(* IEC 61131-3 sources: 1326_JeddahAppartment/1326 - Jeddah Appartment - Last/PLC2, 9 files *)

(* ---- PrgConnectHMIs.ST ---- *)
Type
  T_HMI_Info : struct
     SNo          : USINT;
     readStAdd    : UINT;
     writeStAdd   : UINT;
     readNoPoint  : UINT;
     writeNoPoint : UINT;
  End_Struct;

  //================= Read from HMI =================

  TShutterControl : struct
     Dw : WORD;
     UP : WORD;
  End_Struct;

  TFCU_Control : struct
     onOff       : WORD;
     SetTempCtrl : WORD; //  bit 0 for increment, bit 1 for decrement
     setTemp     : INT;
     fanSpeed    : WORD;
     mode        : WORD;
  End_Struct;

  T_HMI_DataRead : struct
     enLights   : Array[1..17] of WORD;
     enOutlets  : Array[1..8] of WORD;
     enShutters : Array[1..6] of TShutterControl;
     enFCUs     : Array[1..3] of TFCU_Control;
  End_Struct;

  //================= Write To HMI ==================

  TShutterStatus : struct
     Dw  : WORD;
     UP  : WORD;
     pos : WORD;
  End_Struct;

  TFCU_Status  : Struct
     onOffStatus    : WORD;
     setTemp        : INT;
     roomTemp       : INT;
     fanSpeed       : WORD;
     mode           : WORD;
     valve          : WORD;
     fanSpeedCtrl   : WORD;
     fanRotationVar : WORD;   // var for rotating the fan GIF in the HMI according to the current fan speed
  End_Struct;

  T_HMI_DataWrite : struct
     lightsStatus     : Array[1..17] of WORD;
     outletsStatus    : Array[1..8]  of WORD;
     motionSensStatus : Array[1..4]  of WORD;
     shuttersStatus   : Array[1..6]  of TShutterStatus;
     FCUs_Status      : Array[1..3]  of TFCU_Status;
  End_Struct;

End_Type

Var_Global Constant
   numOfHMIs : INT := 11;
End_Var

Var_Global Retain
   HMIs_DataRead  : Array[1..numOfHMIs] of T_HMI_DataRead;     // Data is read from HMI
   HMIs_DataWrite : Array[1..numOfHMIs] of T_HMI_DataWrite;    // Data is written to HMI

   HMIs_Info : Array[1..numOfHMIs] of T_HMI_Info := [()];
End_Var

Var_Global
  cmdArr : Array[1..numOfHMIs * 2] of TCmdStruct;
  GrSel  : USINT ;
End_Var

PROGRAM PrgConnectHMIs
  VAR_INPUT
  END_VAR
  VAR_OUTPUT
  END_VAR
  VAR
  master : fbModbusRTUmas2;
  //cmdArr : Array[1..numOfHMIs * 2] of TCmdStruct;

  i      : INT ;
  maxCmd : USINT;

  END_VAR
  VAR_TEMP
  END_VAR

  if IS_COLD_RESTART_PLC or IS_HOT_RESTART_PLC then
     GrSel := 2;
  end_if;

  for i := 1 to numOfHMIs do
      ModbusCmd(Gr := 2, SNo := HMIs_Info[i].SNo, FNC := 3,  StAdr := HMIs_Info[i].readStAdd,   NoPoint := HMIs_Info[i].readNoPoint, PtrData := adr(HMIs_DataRead[i]), Cmd := cmdArr[i*2-1]) ;

      ModbusCmd(Gr := 2, SNo := HMIs_Info[i].SNo, FNC := 16, StAdr := HMIs_Info[i].writeStAdd , NoPoint := HMIs_Info[i].writeNoPoint, PtrData := adr(HMIs_DataWrite[i]), Cmd := cmdArr[i*2]) ;
  end_for;

  //maxCmd := INT_TO_USINT(numOfHMIs * 2);

  maxCmd := 2;
  master(EN := true, GrSel := GrSel,  MaxCmd := maxCmd , chanCode := CH2_uni , Delay := T#0.2s, Commands := cmdArr[1], MBtimeOut := T#0.5s);

END_PROGRAM

(* ---- PrgDiningRoom.ST ---- *)
VAR_GLOBAL CONSTANT
   NumOfLightDiningRoom      : USINT := 5;
   NumOfOutletDiningRoom     : USINT := 2;
   NumOfCurtainDiningRoom    : USINT := 0;
   NumOfMotionSensDiningRoom : USINT := 1;
   NumOfFCUsDiningRoom       : USINT := 1;
   NumOfHMIsDiningRoom       : USINT := 2;
END_VAR

VAR_GLOBAL RETAIN
   lightsStatusDiningRoom  {PUBLIC_API} : TLightsStatus;
   outletsStatusDiningRoom {PUBLIC_API} : TOutletsStatus;
   setTempFCU_DiningRoom  : Array[1..NumOfFCUsDiningRoom] of REAL := [20];

END_VAR

PROGRAM PrgDiningRoom

  VAR
  //WebMaker
  lightsSelect   : BOOL;
  socketsSelect  : BOOL;
  shuttersSelect : BOOL;
  AC_Select      : BOOL;
  navSelect      : usint;

  //RCU
  RCU_ethAdr   : TRemoteEthAdr;
  RCU_IP : TIPadr := [192, 168, 0, 23];
  RCU_Ch_localPort : UINT;
  Set_IP           : BOOL;
  GetAllStatus  : BOOL;
  SendIamServer : BOOL;

  //controlRoom
  controlRoom   : fbControlRoom ;
  lightsOutputDevs     : TlightsOutputDevs     := [(DevAddress := 1 , loopAddress := 1),(DevAddress := 1 , loopAddress := 2),
                                                   (DevAddress := 1 , loopAddress := 3),(DevAddress := 1 , loopAddress := 4),
                                                   (DevAddress := 1 , loopAddress := 5)];

  outletOutputDevs     : ToutletOutputDevs     := [(DevAddress := 1 , loopAddress := 6),(DevAddress := 1 , loopAddress := 7)];

  (*curtainsUpOutputDevs : TcurtainsUpOutputDevs := [(DevAddress := 1 , loopAddress := 8)];
  curtainsDwOutputDevs : TcurtainsDwOutputDevs := [(DevAddress := 1 , loopAddress := 9)]; *)

  motionSensOutputDevs : TMotionSensOutputDevs := [(DevAddress := 1 , loopAddress := 1)];

  EnLights                            : TEnLights     ;
  EnLightsAN       {PUBLIC_API}       : TEnLightsAN   ;
  EnOutlets                           : TEnOutlets    ;
  EnOutletsAN      {PUBLIC_API}       : TEnOutletsAN  ;
  EnCurtainsUp     {PUBLIC_API}       : TEnCurtainsUp ;
  EnCurtainsDw     {PUBLIC_API}       : TEnCurtainsDW ;
   //EnLightsDiningRoomAN1  {PUBLIC_API}      : TEnLightsAN1    ;
   //stLightsDiningRoomAN  {PUBLIC_API}       : BOOL     ;
  //curtainsFB       : TCurtainsFB;
  //CurtainPositWm   : TCurtainPositWm;

  //
  enLights_RT  : Array[1..NumOfHMIsDiningRoom,1..NumOfLightDiningRoom] of R_TRIG;
  enLights_FT  : Array[1..NumOfHMIsDiningRoom,1..NumOfLightDiningRoom] of F_TRIG;

  enOutlets_RT : Array[1..NumOfHMIsDiningRoom,1..NumOfOutletDiningRoom] of R_TRIG;
  enOutlets_FT : Array[1..NumOfHMIsDiningRoom,1..NumOfOutletDiningRoom] of F_TRIG;

  (*
  enCurtainsUP_RT : Array[1..NumOfHMIsDiningRoom,1..NumOfCurtainDiningRoom] of R_TRIG;
  enCurtainsUP_FT : Array[1..NumOfHMIsDiningRoom,1..NumOfCurtainDiningRoom] of F_TRIG;

  enCurtainsDW_RT : Array[1..NumOfHMIsDiningRoom,1..NumOfCurtainDiningRoom] of R_TRIG;
  enCurtainsDW_FT : Array[1..NumOfHMIsDiningRoom,1..NumOfCurtainDiningRoom] of F_TRIG;
  *)

  //
  i , j : USINT;
  afterRestart_TP : TP;
  afterRestart_TP_FT : F_TRIG;

  //
  motionSensStatus                : TMotionSensStatus;
  CurtainsUpStatus   {PUBLIC_API} : TCurtainsUpStatus;
  CurtainsDwStatus   {PUBLIC_API} : TCurtainsDwStatus;

  // FCU VARS
  FCU          : Array[1..NumOfFCUsDiningRoom] of fbControlFCU;
  enableFCU    : Array[1..NumOfFCUsDiningRoom] of BOOL;
  settingsFCU  : Array[1..NumOfFCUsDiningRoom] of TFCU_Settings;

  //modeFCU      : Array[1..NumOfFCUsDiningRoom] of TFCU_Mode;
  //fanSpeedFCU  : Array[1..NumOfFCUsDiningRoom] of TFCU_FanSpeed;

  enFCUs_FT    : Array[1..NumOfHMIsDiningRoom,1..NumOfFCUsDiningRoom] of F_TRIG;
  enFCUs_RT    : Array[1..NumOfHMIsDiningRoom,1..NumOfFCUsDiningRoom] of R_TRIG;

  enFanHigh_RT : Array[1..NumOfHMIsDiningRoom,1..NumOfFCUsDiningRoom] of R_TRIG;
  enFanMed_RT  : Array[1..NumOfHMIsDiningRoom,1..NumOfFCUsDiningRoom] of R_TRIG;
  enFanLow_RT  : Array[1..NumOfHMIsDiningRoom,1..NumOfFCUsDiningRoom] of R_TRIG;
  enFanAuto_RT : Array[1..NumOfHMIsDiningRoom,1..NumOfFCUsDiningRoom] of R_TRIG;

  enFCUCool_RT    : Array[1..NumOfHMIsDiningRoom,1..NumOfFCUsDiningRoom] of R_TRIG;
  enFCUFanOnly_RT : Array[1..NumOfHMIsDiningRoom,1..NumOfFCUsDiningRoom] of R_TRIG;

  enSetTempIncr_RT : Array[1..NumOfHMIsDiningRoom,1..NumOfFCUsDiningRoom] of R_TRIG;
  enSetTempIncr_FT : Array[1..NumOfHMIsDiningRoom,1..NumOfFCUsDiningRoom] of F_TRIG;

  enSetTempDecr_RT : Array[1..NumOfHMIsDiningRoom,1..NumOfFCUsDiningRoom] of R_TRIG;
  enSetTempDecr_FT : Array[1..NumOfHMIsDiningRoom,1..NumOfFCUsDiningRoom] of F_TRIG;

  //HMIs[1..num
  HMI_Index : USINT;
  RCU_Index : USINT;
  HMI_Addresses : Array[1..NumOfHMIsDiningRoom] of USINT := [2, 10];

  END_VAR

   if navSelect = 0 then
     lightsSelect   := 1;
     socketsSelect  := 0;
     AC_Select      := 0;
  elsif navSelect = 1 then
     lightsSelect   := 0;
     socketsSelect  := 1;
     AC_Select      := 0;
  elsif navSelect = 2 then
     lightsSelect   := 0;
     socketsSelect  := 0;
     AC_Select      := 1;
  end_if;

  HMI_Index := 2;
  RCU_Index := 2;

  if GetRemoteIPaddress(chanCode := Eth1_uni1, ethAdr := RCU_ethAdr) then
     RCUs_IPs[RCU_Index] := RCU_ethAdr.remoteIP;
  end_if;

  HMIs_Info[HMI_Index].SNo := HMI_Addresses[1];
  HMIs_Info[HMI_Index].readStAdd  := 261;
  HMIs_Info[HMI_Index].writeStAdd := 321;
  HMIs_Info[HMI_Index].readNoPoint  := SIZEOF(HMIs_DataRead[HMI_Index]) / 2;
  HMIs_Info[HMI_Index].writeNoPoint := SIZEOF(HMIs_DataWrite[HMI_Index]) / 2;

  for i := 1 to NumOfHMIsDiningRoom-1 do
    HMIs_Info[HMI_Index+i] := HMIs_Info[HMI_Index];
    HMIs_Info[HMI_Index+i].SNo := HMI_Addresses[i+1];
  end_for;

  afterRestart_TP(IN := IS_COLD_RESTART_PLC or IS_HOT_RESTART_PLC, PT := T#2s );
  afterRestart_TP_FT(CLK := afterRestart_TP.Q);

  if afterRestart_TP_FT.Q then
     SendIamServer := 1;
  end_if;

  controlRoom(RCU_ChCode := ETH1_uni1 , RCU_PingDone := RCUs_PingDone[RCU_Index],
              numOfLights := NumOfLightDiningRoom , numOfOutlets := NumOfOutletDiningRoom , numOfCurtains := NumOfCurtainDiningRoom, numOfMotionSens := NumOfMotionSensDiningRoom,
              lightsOutputDevs := lightsOutputDevs , outletOutputDevs := outletOutputDevs ,
              RCU_CH_IN := void(ETH1_uni1_IN) , LightsStatus := lightsStatusDiningRoom ,OutletsStatus := outletsStatusDiningRoom, MotionSenStatus := motionSensStatus,
              EnLights := EnLights , EnLightsAN := EnLightsAN , EnOutlets := EnOutlets ,EnOutletsAN :=EnOutletsAN ,
              SendIamServer := SendIamServer , GetAllStatus := GetAllStatus);

              //stLightsDiningRoomAN := lightsStatusDiningRoom[1];

   FCU[1](enable := enableFCU[1], mode := settingsFCU[1].FCU_Mode, fanSpeed := settingsFCU[1].FCU_FanSpeed, setTemp := setTempFCU_DiningRoom[1], temp := FCU_Temp_DiningRoom, valve := FCU_valve_DiningRoom, fanLow := FCU_fanLow_DiningRoom,
                 fanMed := FCU_fanMed_DiningRoom, fanHigh := FCU_fanHigh_DiningRoom);

   for i := 1 to NumOfLightDiningRoom do
       HMIs_DataWrite[HMI_Index].lightsStatus[i] := BOOL_TO_WORD(lightsStatusDiningRoom[i]);
   end_for;

   for i := 1 to NumOfOutletDiningRoom do
       HMIs_DataWrite[HMI_Index].outletsStatus[i] := BOOL_TO_WORD(outletsStatusDiningRoom[i]);
   end_for;

   for i := 1 to NumOfMotionSensDiningRoom do
       HMIs_DataWrite[HMI_Index].motionSensStatus[i] := BOOL_TO_WORD(motionSensStatus[i]);
   end_for;

   for i := 1 to NumOfFCUsDiningRoom do
      HMIs_DataWrite[HMI_Index].FCUs_Status[i] := FCU[i].FCU_Status;
   end_for;

   for i := 1 to NumOfHMIsDiningRoom-1 do
     HMIs_DataWrite[HMI_Index+i] := HMIs_DataWrite[HMI_Index];
   end_for;

   for j := 1 to NumOfHMIsDiningRoom do
     for i := 1 to NumOfLightDiningRoom do

         enLights_RT[j,i](CLK := HMIs_DataRead[HMI_Index + j - 1].enLights[i]);

         enLights_FT[j,i](CLK := HMIs_DataRead[HMI_Index + j - 1].enLights[i]);

         if enLights_RT[j,i].Q or enLights_FT[j,i].Q then
            EnLights[i] := 1;
         end_if;
     end_for;
   end_for;

   for j := 1 to NumOfHMIsDiningRoom do
     for i := 1 to NumOfOutletDiningRoom do

         enOutlets_RT[j,i](CLK := HMIs_DataRead[HMI_Index + j - 1].enOutlets[i]);

         enOutlets_FT[j,i](CLK := HMIs_DataRead[HMI_Index + j - 1].enOutlets[i]);

         if enOutlets_RT[j,i].Q or enOutlets_FT[j,i].Q then
            EnOutlets[i] := 1;
         end_if;
     end_for;
   end_for;

  (*
   for j := 1 to NumOfHMIsDiningRoom do
     for i := 1 to NumOfCurtainDiningRoom do

         enCurtainsUP_RT[j,i](CLK := HMIs_DataRead[HMI_Index + j - 1].enShutters[i].UP.0);

         enCurtainsUP_FT[j,i](CLK := HMIs_DataRead[HMI_Index + j - 1].enShutters[i].UP.0);

         if enCurtainsUP_RT[j,i].Q or enCurtainsUP_FT[j,i].Q then
            EnCurtainsUp[i] := 1;
         end_if;

         enCurtainsDW_RT[j,i](CLK := HMIs_DataRead[HMI_Index + j - 1].enShutters[i].Dw.0);

         enCurtainsDW_FT[j,i](CLK := HMIs_DataRead[HMI_Index + j - 1].enShutters[i].Dw.0);

         if enCurtainsDW_RT[j,i].Q or enCurtainsDW_FT[j,i].Q then
            EnCurtainsDw[i] := 1;
         end_if;

     end_for;
   end_for;*)

   for j := 1 to NumOfHMIsDiningRoom do
      for i := 1 to NumOfFCUsDiningRoom do
          enFCUs_FT[j,i](CLK := HMIs_DataRead[HMI_Index + j - 1].enFCUs[i].onOff);
          enFCUs_RT[j,i](CLK := HMIs_DataRead[HMI_Index + j - 1].enFCUs[i].onOff);

          if enFCUs_FT[j,i].Q then
             enableFCU[i] := 0;
          end_if;
          if enFCUs_RT[j,i].Q then
             enableFCU[i] := 1;
          end_if;

          enFanAuto_RT[j,i](CLK := (HMIs_DataRead[HMI_Index + j - 1].enFCUs[i].fanSpeed = 8));
          enFanLow_RT[j,i](CLK := HMIs_DataRead[HMI_Index + j - 1].enFCUs[i].fanSpeed.0);
          enFanMed_RT[j,i](CLK := HMIs_DataRead[HMI_Index + j - 1].enFCUs[i].fanSpeed.1);
          enFanHigh_RT[j,i](CLK := HMIs_DataRead[HMI_Index + j - 1].enFCUs[i].fanSpeed.2);

          if enFanAuto_RT[j,i].Q then
             settingsFCU[i].FCU_FanSpeed := auto;
          end_if;
          if enFanLow_RT[j,i].Q then
             settingsFCU[i].FCU_FanSpeed := low;
          end_if;
          if enFanMed_RT[j,i].Q then
             settingsFCU[i].FCU_FanSpeed := med;
          end_if;
          if enFanHigh_RT[j,i].Q then
             settingsFCU[i].FCU_FanSpeed := high;
          end_if;

          enFCUCool_RT[j,i](CLK := (HMIs_DataRead[HMI_Index + j - 1].enFCUs[i].mode = 0));
          enFCUFanOnly_RT[j,i](CLK := HMIs_DataRead[HMI_Index + j - 1].enFCUs[i].mode.0);

          if enFCUCool_RT[j,i].Q then
             settingsFCU[i].FCU_Mode := cooling;
          end_if;
          if enFCUFanOnly_RT[j,i].Q then
             settingsFCU[i].FCU_Mode := fanOnly;
          end_if;

          enSetTempIncr_RT[j,i](CLK := HMIs_DataRead[HMI_Index + j - 1].enFCUs[i].SetTempCtrl.0);
          enSetTempIncr_FT[j,i](CLK := HMIs_DataRead[HMI_Index + j - 1].enFCUs[i].SetTempCtrl.0);

          if enSetTempIncr_RT[j,i].Q or enSetTempIncr_FT[j,i].Q then
             setTempFCU_DiningRoom[j] := setTempFCU_DiningRoom[j] + 0.5;
          end_if;

          enSetTempDecr_RT[j,i](CLK := HMIs_DataRead[HMI_Index + j - 1].enFCUs[i].SetTempCtrl.1);
          enSetTempDecr_FT[j,i](CLK := HMIs_DataRead[HMI_Index + j - 1].enFCUs[i].SetTempCtrl.1);

          if enSetTempDecr_RT[j,i].Q or enSetTempDecr_FT[j,i].Q then
             setTempFCU_DiningRoom[j] := setTempFCU_DiningRoom[j] - 0.5;
          end_if;

      end_for;
   end_for;

END_PROGRAM

(* ---- PrgInterance.ST ---- *)
VAR_GLOBAL CONSTANT
   NumOfLightInter    :USINT := 6;
   NumOfOutletInter   :USINT := 1;
   NumOfCurtainInter  :USINT := 0;
END_VAR

VAR_GLOBAL RETAIN
   lightsStatusInter  : TLightsStatus;
   outletsStatusInter : TOutletsStatus;
END_VAR

PROGRAM PrgInterance

  VAR
  //WebMaker
  lightsSelect   : BOOL;
  socketsSelect  : BOOL;
  navSelect      : usint;

  //RCU
  RCU_ethAdrToSet   : TRemoteEthAdr;
  RCU_IP : TIPadr := [192, 168, 0, 24];
  RCU_Ch_localPort : UINT;
  Set_IP           : BOOL;
  GetAllStatus  : BOOL;
  SendIamServer : BOOL;

  //controlRoom
 // controlRoom   : fbControlRoom ;
  lightsOutputDevs     : TlightsOutputDevs     := [(DevAddress := 1 , loopAddress := 1),(DevAddress := 1 , loopAddress := 2),
                                                   (DevAddress := 1 , loopAddress := 3),(DevAddress := 1 , loopAddress := 4),
                                                   (DevAddress := 1 , loopAddress := 5),(DevAddress := 1 , loopAddress := 6)];
  outletOutputDevs     : ToutletOutputDevs     := [(DevAddress := 1 , loopAddress := 7)];

  EnLights         : TEnLights     ;
  EnOutlets        : TEnOutlets    ;
  EnCurtainsUp     : TEnCurtainsUp ;
  EnCurtainsDw     : TEnCurtainsDW ;
  curtainsFB       : TCurtainsFB;
  CurtainsUpStatus : TCurtainsUpStatus;
  CurtainsDwStatus : TCurtainsDwStatus;
  END_VAR

  if navSelect = 0 then
     lightsSelect   := 1;
     socketsSelect  := 0;

  elsif navSelect = 1 then
     lightsSelect   := 0;
     socketsSelect  := 1;
  end_if;

  RCU_Ch_localPort := 61000;
  RCU_ethAdrToSet.remotePort := 3341;
  RCU_ethAdrToSet.localPort  := RCU_Ch_localPort;
  RCU_ethAdrToSet.remoteIP   := RCU_IP;

 (* controlRoom(RCU_ChCode := ETH1_uni0 , RCU_IP_toSet := RCU_IP, RCU_ethAdrToSet := RCU_ethAdrToSet ,
              numOfLights := NumOfLightInter , numOfOutlets := NumOfOutletInter , numOfCurtains := NumOfCurtainInter,
              lightsOutputDevs := lightsOutputDevs , outletOutputDevs := outletOutputDevs ,
              RCU_CH_IN := void(ETH1_uni0_IN) , LightsStatus := lightsStatusInter , OutletsStatus := outletsStatusInter,
              CurtainsUpStatus :=CurtainsUpStatus ,CurtainsDwStatus := CurtainsDwStatus ,CurtainsFB :=curtainsFB ,
              EnLights := EnLights , EnOutlets := EnOutlets ,EnCurtainsUp := EnCurtainsUp ,EnCurtainsDw :=EnCurtainsDw,
              SendIamServer := SendIamServer , GetAllStatus := GetAllStatus); *)
END_PROGRAM

(* ---- PrgKitchen.ST ---- *)
VAR_GLOBAL CONSTANT
   NumOfLightKitchen      : USINT := 4;
   NumOfOutletKitchen     : USINT := 5;
   NumOfCurtainKitchen    : USINT := 0;
   NumOfMotionSensKitchen : USINT := 1;
   NumOfFCUsKitchen       : USINT := 1;
   NumOfHMIsKitchen       : USINT := 1;
END_VAR

VAR_GLOBAL RETAIN
   lightsStatusKitchen  {PUBLIC_API} : TLightsStatus;
   outletsStatusKitchen {PUBLIC_API} : TOutletsStatus;
   setTempFCU_Kitchen  : Array[1..NumOfFCUsKitchen] of REAL := [20];

END_VAR

PROGRAM PrgKitchen

  VAR
  //WebMaker
  lightsSelect   : BOOL;
  socketsSelect  : BOOL;
  shuttersSelect : BOOL;
  AC_Select      : BOOL;
  navSelect      : usint;

  //RCU
  RCU_ethAdr   : TRemoteEthAdr;
  RCU_IP : TIPadr := [192, 168, 0, 23];
  RCU_Ch_localPort : UINT;
  Set_IP           : BOOL;
  GetAllStatus  : BOOL;
  SendIamServer : BOOL;

  //controlRoom
  controlRoom   : fbControlRoom ;
  lightsOutputDevs     : TlightsOutputDevs     := [(DevAddress := 1 , loopAddress := 1),(DevAddress := 1 , loopAddress := 2),
                                                   (DevAddress := 1 , loopAddress := 3),(DevAddress := 1 , loopAddress := 4)];

  outletOutputDevs     : ToutletOutputDevs     := [(DevAddress := 1 , loopAddress := 5),(DevAddress := 1 , loopAddress := 6),
                                                   (DevAddress := 1 , loopAddress := 7),(DevAddress := 1 , loopAddress := 8),(DevAddress := 1 , loopAddress := 9)];

  (*curtainsUpOutputDevs : TcurtainsUpOutputDevs := [(DevAddress := 1 , loopAddress := 8)];
  curtainsDwOutputDevs : TcurtainsDwOutputDevs := [(DevAddress := 1 , loopAddress := 9)]; *)

  motionSensOutputDevs : TMotionSensOutputDevs := [(DevAddress := 1 , loopAddress := 1)];

  EnLights                            : TEnLights     ;
  EnLightsAN       {PUBLIC_API}       : TEnLightsAN   ;
  EnOutlets                           : TEnOutlets    ;
  EnOutletsAN      {PUBLIC_API}       : TEnOutletsAN  ;
  EnCurtainsUp     {PUBLIC_API}       : TEnCurtainsUp ;
  EnCurtainsDw     {PUBLIC_API}       : TEnCurtainsDW ;
   //EnLightsKitchenAN1  {PUBLIC_API}      : TEnLightsAN1    ;
   //stLightsKitchenAN  {PUBLIC_API}       : BOOL     ;
  //curtainsFB       : TCurtainsFB;
  //CurtainPositWm   : TCurtainPositWm;

  //
  enLights_RT  : Array[1..NumOfHMIsKitchen,1..NumOfLightKitchen] of R_TRIG;
  enLights_FT  : Array[1..NumOfHMIsKitchen,1..NumOfLightKitchen] of F_TRIG;

  enOutlets_RT : Array[1..NumOfHMIsKitchen,1..NumOfOutletKitchen] of R_TRIG;
  enOutlets_FT : Array[1..NumOfHMIsKitchen,1..NumOfOutletKitchen] of F_TRIG;

  (*
  enCurtainsUP_RT : Array[1..NumOfHMIsKitchen,1..NumOfCurtainKitchen] of R_TRIG;
  enCurtainsUP_FT : Array[1..NumOfHMIsKitchen,1..NumOfCurtainKitchen] of F_TRIG;

  enCurtainsDW_RT : Array[1..NumOfHMIsKitchen,1..NumOfCurtainKitchen] of R_TRIG;
  enCurtainsDW_FT : Array[1..NumOfHMIsKitchen,1..NumOfCurtainKitchen] of F_TRIG;
  *)

  //
  i , j : USINT;
  afterRestart_TP : TP;
  afterRestart_TP_FT : F_TRIG;

  //
  motionSensStatus                : TMotionSensStatus;
  CurtainsUpStatus   {PUBLIC_API} : TCurtainsUpStatus;
  CurtainsDwStatus   {PUBLIC_API} : TCurtainsDwStatus;

  // FCU VARS
  FCU          : Array[1..NumOfFCUsKitchen] of fbControlFCU;
  enableFCU    : Array[1..NumOfFCUsKitchen] of BOOL;
  settingsFCU  : Array[1..NumOfFCUsKitchen] of TFCU_Settings;

  //modeFCU      : Array[1..NumOfFCUsKitchen] of TFCU_Mode;
  //fanSpeedFCU  : Array[1..NumOfFCUsKitchen] of TFCU_FanSpeed;

  enFCUs_FT    : Array[1..NumOfHMIsKitchen,1..NumOfFCUsKitchen] of F_TRIG;
  enFCUs_RT    : Array[1..NumOfHMIsKitchen,1..NumOfFCUsKitchen] of R_TRIG;

  enFanHigh_RT : Array[1..NumOfHMIsKitchen,1..NumOfFCUsKitchen] of R_TRIG;
  enFanMed_RT  : Array[1..NumOfHMIsKitchen,1..NumOfFCUsKitchen] of R_TRIG;
  enFanLow_RT  : Array[1..NumOfHMIsKitchen,1..NumOfFCUsKitchen] of R_TRIG;
  enFanAuto_RT : Array[1..NumOfHMIsKitchen,1..NumOfFCUsKitchen] of R_TRIG;

  enFCUCool_RT    : Array[1..NumOfHMIsKitchen,1..NumOfFCUsKitchen] of R_TRIG;
  enFCUFanOnly_RT : Array[1..NumOfHMIsKitchen,1..NumOfFCUsKitchen] of R_TRIG;

  enSetTempIncr_RT : Array[1..NumOfHMIsKitchen,1..NumOfFCUsKitchen] of R_TRIG;
  enSetTempIncr_FT : Array[1..NumOfHMIsKitchen,1..NumOfFCUsKitchen] of F_TRIG;

  enSetTempDecr_RT : Array[1..NumOfHMIsKitchen,1..NumOfFCUsKitchen] of R_TRIG;
  enSetTempDecr_FT : Array[1..NumOfHMIsKitchen,1..NumOfFCUsKitchen] of F_TRIG;

  //HMIs[1..num
  HMI_Index : USINT;
  RCU_Index : USINT;
  HMI_Addresses : Array[1..NumOfHMIsKitchen] of USINT := [7];

  END_VAR

     if navSelect = 0 then
     lightsSelect   := 1;
     socketsSelect  := 0;
     AC_Select      := 0;
  elsif navSelect = 1 then
     lightsSelect   := 0;
     socketsSelect  := 1;
     AC_Select      := 0;
  elsif navSelect = 2 then
     lightsSelect   := 0;
     socketsSelect  := 0;
     AC_Select      := 1;
  end_if;

  HMI_Index := 6;
  RCU_Index := 4;

  if GetRemoteIPaddress(chanCode := Eth1_uni3, ethAdr := RCU_ethAdr) then
     RCUs_IPs[RCU_Index] := RCU_ethAdr.remoteIP;
  end_if;

  HMIs_Info[HMI_Index].SNo := HMI_Addresses[1];
  HMIs_Info[HMI_Index].readStAdd  := 521;
  HMIs_Info[HMI_Index].writeStAdd := 581;
  HMIs_Info[HMI_Index].readNoPoint  := SIZEOF(HMIs_DataRead[HMI_Index]) / 2;
  HMIs_Info[HMI_Index].writeNoPoint := SIZEOF(HMIs_DataWrite[HMI_Index]) / 2;

  for i := 1 to NumOfHMIsKitchen-1 do
    HMIs_Info[HMI_Index+i] := HMIs_Info[HMI_Index];
    HMIs_Info[HMI_Index+i].SNo := HMI_Addresses[i+1];
  end_for;

  afterRestart_TP(IN := IS_COLD_RESTART_PLC or IS_HOT_RESTART_PLC, PT := T#2s );
  afterRestart_TP_FT(CLK := afterRestart_TP.Q);

  if afterRestart_TP_FT.Q then
     SendIamServer := 1;
  end_if;

  controlRoom(RCU_ChCode := ETH1_uni3 , RCU_PingDone := RCUs_PingDone[RCU_Index],
              numOfLights := NumOfLightKitchen , numOfOutlets := NumOfOutletKitchen , numOfCurtains := NumOfCurtainKitchen, numOfMotionSens := NumOfMotionSensKitchen,
              lightsOutputDevs := lightsOutputDevs , outletOutputDevs := outletOutputDevs ,
              RCU_CH_IN := void(ETH1_uni3_IN) , LightsStatus := lightsStatusKitchen ,OutletsStatus := outletsStatusKitchen, MotionSenStatus := motionSensStatus,
              EnLights := EnLights , EnLightsAN := EnLightsAN , EnOutlets := EnOutlets ,EnOutletsAN :=EnOutletsAN ,
              SendIamServer := SendIamServer , GetAllStatus := GetAllStatus);

              //stLightsKitchenAN := lightsStatusKitchen[1];

   FCU[1](enable := enableFCU[1], mode := settingsFCU[1].FCU_Mode, fanSpeed := settingsFCU[1].FCU_FanSpeed, setTemp := setTempFCU_Kitchen[1], temp := FCU_Temp_Kitchen, valve := FCU_valve_Kitchen, fanLow := FCU_fanLow_Kitchen,
                 fanMed := FCU_fanMed_Kitchen, fanHigh := FCU_fanHigh_Kitchen);

   for i := 1 to NumOfLightKitchen do
       HMIs_DataWrite[HMI_Index].lightsStatus[i] := BOOL_TO_WORD(lightsStatusKitchen[i]);
   end_for;

   for i := 1 to NumOfOutletKitchen do
       HMIs_DataWrite[HMI_Index].outletsStatus[i] := BOOL_TO_WORD(outletsStatusKitchen[i]);
   end_for;

   for i := 1 to NumOfMotionSensKitchen do
       HMIs_DataWrite[HMI_Index].motionSensStatus[i] := BOOL_TO_WORD(motionSensStatus[i]);
   end_for;

   for i := 1 to NumOfFCUsKitchen do
      HMIs_DataWrite[HMI_Index].FCUs_Status[i] := FCU[i].FCU_Status;
   end_for;

   for i := 1 to NumOfHMIsKitchen-1 do
     HMIs_DataWrite[HMI_Index+i] := HMIs_DataWrite[HMI_Index];
   end_for;

   for j := 1 to NumOfHMIsKitchen do
     for i := 1 to NumOfLightKitchen do

         enLights_RT[j,i](CLK := HMIs_DataRead[HMI_Index + j - 1].enLights[i]);

         enLights_FT[j,i](CLK := HMIs_DataRead[HMI_Index + j - 1].enLights[i]);

         if enLights_RT[j,i].Q or enLights_FT[j,i].Q then
            EnLights[i] := 1;
         end_if;
     end_for;
   end_for;

   for j := 1 to NumOfHMIsKitchen do
     for i := 1 to NumOfOutletKitchen do

         enOutlets_RT[j,i](CLK := HMIs_DataRead[HMI_Index + j - 1].enOutlets[i]);

         enOutlets_FT[j,i](CLK := HMIs_DataRead[HMI_Index + j - 1].enOutlets[i]);

         if enOutlets_RT[j,i].Q or enOutlets_FT[j,i].Q then
            EnOutlets[i] := 1;
         end_if;
     end_for;
   end_for;

  (*
   for j := 1 to NumOfHMIsKitchen do
     for i := 1 to NumOfCurtainKitchen do

         enCurtainsUP_RT[j,i](CLK := HMIs_DataRead[HMI_Index + j - 1].enShutters[i].UP.0);

         enCurtainsUP_FT[j,i](CLK := HMIs_DataRead[HMI_Index + j - 1].enShutters[i].UP.0);

         if enCurtainsUP_RT[j,i].Q or enCurtainsUP_FT[j,i].Q then
            EnCurtainsUp[i] := 1;
         end_if;

         enCurtainsDW_RT[j,i](CLK := HMIs_DataRead[HMI_Index + j - 1].enShutters[i].Dw.0);

         enCurtainsDW_FT[j,i](CLK := HMIs_DataRead[HMI_Index + j - 1].enShutters[i].Dw.0);

         if enCurtainsDW_RT[j,i].Q or enCurtainsDW_FT[j,i].Q then
            EnCurtainsDw[i] := 1;
         end_if;

     end_for;
   end_for;*)

   for j := 1 to NumOfHMIsKitchen do
      for i := 1 to NumOfFCUsKitchen do
          enFCUs_FT[j,i](CLK := HMIs_DataRead[HMI_Index + j - 1].enFCUs[i].onOff);
          enFCUs_RT[j,i](CLK := HMIs_DataRead[HMI_Index + j - 1].enFCUs[i].onOff);

          if enFCUs_FT[j,i].Q then
             enableFCU[i] := 0;
          end_if;
          if enFCUs_RT[j,i].Q then
             enableFCU[i] := 1;
          end_if;

          enFanAuto_RT[j,i](CLK := (HMIs_DataRead[HMI_Index + j - 1].enFCUs[i].fanSpeed = 8));
          enFanLow_RT[j,i](CLK := HMIs_DataRead[HMI_Index + j - 1].enFCUs[i].fanSpeed.0);
          enFanMed_RT[j,i](CLK := HMIs_DataRead[HMI_Index + j - 1].enFCUs[i].fanSpeed.1);
          enFanHigh_RT[j,i](CLK := HMIs_DataRead[HMI_Index + j - 1].enFCUs[i].fanSpeed.2);

          if enFanAuto_RT[j,i].Q then
             settingsFCU[i].FCU_FanSpeed := auto;
          end_if;
          if enFanLow_RT[j,i].Q then
             settingsFCU[i].FCU_FanSpeed := low;
          end_if;
          if enFanMed_RT[j,i].Q then
             settingsFCU[i].FCU_FanSpeed := med;
          end_if;
          if enFanHigh_RT[j,i].Q then
             settingsFCU[i].FCU_FanSpeed := high;
          end_if;

          enFCUCool_RT[j,i](CLK := (HMIs_DataRead[HMI_Index + j - 1].enFCUs[i].mode = 0));
          enFCUFanOnly_RT[j,i](CLK := HMIs_DataRead[HMI_Index + j - 1].enFCUs[i].mode.0);

          if enFCUCool_RT[j,i].Q then
             settingsFCU[i].FCU_Mode := cooling;
          end_if;
          if enFCUFanOnly_RT[j,i].Q then
             settingsFCU[i].FCU_Mode := fanOnly;
          end_if;

          enSetTempIncr_RT[j,i](CLK := HMIs_DataRead[HMI_Index + j - 1].enFCUs[i].SetTempCtrl.0);
          enSetTempIncr_FT[j,i](CLK := HMIs_DataRead[HMI_Index + j - 1].enFCUs[i].SetTempCtrl.0);

          if enSetTempIncr_RT[j,i].Q or enSetTempIncr_FT[j,i].Q then
             setTempFCU_Kitchen[j] := setTempFCU_Kitchen[j] + 0.5;
          end_if;

          enSetTempDecr_RT[j,i](CLK := HMIs_DataRead[HMI_Index + j - 1].enFCUs[i].SetTempCtrl.1);
          enSetTempDecr_FT[j,i](CLK := HMIs_DataRead[HMI_Index + j - 1].enFCUs[i].SetTempCtrl.1);

          if enSetTempDecr_RT[j,i].Q or enSetTempDecr_FT[j,i].Q then
             setTempFCU_Kitchen[j] := setTempFCU_Kitchen[j] - 0.5;
          end_if;

      end_for;
   end_for;

END_PROGRAM

(* ---- PrgLivingRoom.ST ---- *)
VAR_GLOBAL CONSTANT
   NumOfLightLivingRoom      : USINT := 5;
   NumOfOutletLivingRoom     : USINT := 2;
   NumOfCurtainLivingRoom    : USINT := 2;
   NumOfMotionSensLivingRoom : USINT := 1;
   NumOfFCUsLivingRoom       : USINT := 0;
   NumOfHMIsLivingRoom       : USINT := 2;
END_VAR

VAR_GLOBAL RETAIN
   lightsStatusLivingRoom  {PUBLIC_API} : TLightsStatus;
   outletsStatusLivingRoom {PUBLIC_API} : TOutletsStatus;
  // setTempFCU_LivingRoom  : Array[1..NumOfFCUsLivingRoom] of REAL := [20];

END_VAR

PROGRAM PrgLivingRoom

  VAR
  //WebMaker
  lightsSelect   : BOOL;
  socketsSelect  : BOOL;
  shuttersSelect : BOOL;
  AC_Select      : BOOL;
  navSelect      : usint;

  //RCU
  RCU_ethAdr   : TRemoteEthAdr;
  RCU_IP : TIPadr := [192, 168, 0, 23];
  RCU_Ch_localPort : UINT;
  Set_IP           : BOOL;
  GetAllStatus  : BOOL;
  SendIamServer : BOOL;

  //controlRoom
  controlRoom   : fbControlRoom ;
  lightsOutputDevs     : TlightsOutputDevs     := [(DevAddress := 1 , loopAddress := 1),(DevAddress := 1 , loopAddress := 2),
                                                   (DevAddress := 1 , loopAddress := 3),(DevAddress := 1 , loopAddress := 4),
                                                   (DevAddress := 1 , loopAddress := 5)];

  outletOutputDevs     : ToutletOutputDevs     := [(DevAddress := 1 , loopAddress := 6),(DevAddress := 1 , loopAddress := 7)];

  curtainsUpOutputDevs : TcurtainsUpOutputDevs := [(DevAddress := 2 , loopAddress := 1), (DevAddress := 2 , loopAddress := 3)];
  curtainsDwOutputDevs : TcurtainsDwOutputDevs := [(DevAddress := 2 , loopAddress := 2), (DevAddress := 2 , loopAddress := 4)];

  motionSensOutputDevs : TMotionSensOutputDevs := [(DevAddress := 1 , loopAddress := 1)];

  EnLights                            : TEnLights     ;
  EnLightsAN       {PUBLIC_API}       : TEnLightsAN   ;
  EnOutlets                           : TEnOutlets    ;
  EnOutletsAN      {PUBLIC_API}       : TEnOutletsAN  ;
  EnCurtainsUp     {PUBLIC_API}       : TEnCurtainsUp ;
  EnCurtainsDw     {PUBLIC_API}       : TEnCurtainsDW ;
   //EnLightsLivingRoomAN1  {PUBLIC_API}      : TEnLightsAN1    ;
   //stLightsLivingRoomAN  {PUBLIC_API}       : BOOL     ;
  //curtainsFB       : TCurtainsFB;
  //CurtainPositWm   : TCurtainPositWm;

  //
  enLights_RT  : Array[1..NumOfHMIsLivingRoom,1..NumOfLightLivingRoom] of R_TRIG;
  enLights_FT  : Array[1..NumOfHMIsLivingRoom,1..NumOfLightLivingRoom] of F_TRIG;

  enOutlets_RT : Array[1..NumOfHMIsLivingRoom,1..NumOfOutletLivingRoom] of R_TRIG;
  enOutlets_FT : Array[1..NumOfHMIsLivingRoom,1..NumOfOutletLivingRoom] of F_TRIG;

  enCurtainsUP_RT : Array[1..NumOfHMIsLivingRoom,1..NumOfCurtainLivingRoom] of R_TRIG;
  enCurtainsUP_FT : Array[1..NumOfHMIsLivingRoom,1..NumOfCurtainLivingRoom] of F_TRIG;

  enCurtainsDW_RT : Array[1..NumOfHMIsLivingRoom,1..NumOfCurtainLivingRoom] of R_TRIG;
  enCurtainsDW_FT : Array[1..NumOfHMIsLivingRoom,1..NumOfCurtainLivingRoom] of F_TRIG;

  //
  i , j : USINT;
  afterRestart_TP : TP;
  afterRestart_TP_FT : F_TRIG;

  //
  motionSensStatus                : TMotionSensStatus;
  CurtainsUpStatus   {PUBLIC_API} : TCurtainsUpStatus;
  CurtainsDwStatus   {PUBLIC_API} : TCurtainsDwStatus;

  // FCU VARS
 (* FCU          : Array[1..NumOfFCUsLivingRoom] of fbControlFCU;
  enableFCU    : Array[1..NumOfFCUsLivingRoom] of BOOL;
  settingsFCU  : Array[1..NumOfFCUsLivingRoom] of TFCU_Settings;

  //modeFCU      : Array[1..NumOfFCUsLivingRoom] of TFCU_Mode;
  //fanSpeedFCU  : Array[1..NumOfFCUsLivingRoom] of TFCU_FanSpeed;

  enFCUs_FT    : Array[1..NumOfHMIsLivingRoom,1..NumOfFCUsLivingRoom] of F_TRIG;
  enFCUs_RT    : Array[1..NumOfHMIsLivingRoom,1..NumOfFCUsLivingRoom] of R_TRIG;

  enFanHigh_RT : Array[1..NumOfHMIsLivingRoom,1..NumOfFCUsLivingRoom] of R_TRIG;
  enFanMed_RT  : Array[1..NumOfHMIsLivingRoom,1..NumOfFCUsLivingRoom] of R_TRIG;
  enFanLow_RT  : Array[1..NumOfHMIsLivingRoom,1..NumOfFCUsLivingRoom] of R_TRIG;
  enFanAuto_RT : Array[1..NumOfHMIsLivingRoom,1..NumOfFCUsLivingRoom] of R_TRIG;

  enFCUCool_RT    : Array[1..NumOfHMIsLivingRoom,1..NumOfFCUsLivingRoom] of R_TRIG;
  enFCUFanOnly_RT : Array[1..NumOfHMIsLivingRoom,1..NumOfFCUsLivingRoom] of R_TRIG;

  enSetTempIncr_RT : Array[1..NumOfHMIsLivingRoom,1..NumOfFCUsLivingRoom] of R_TRIG;
  enSetTempIncr_FT : Array[1..NumOfHMIsLivingRoom,1..NumOfFCUsLivingRoom] of F_TRIG;

  enSetTempDecr_RT : Array[1..NumOfHMIsLivingRoom,1..NumOfFCUsLivingRoom] of R_TRIG;
  enSetTempDecr_FT : Array[1..NumOfHMIsLivingRoom,1..NumOfFCUsLivingRoom] of F_TRIG;  *)

  //HMIs[1..num
  HMI_Index : USINT;
  RCU_Index : USINT;
  HMI_Addresses : Array[1..NumOfHMIsLivingRoom] of USINT := [3, 5];

  END_VAR

   if navSelect = 0 then
     lightsSelect   := 1;
     socketsSelect  := 0;
     shuttersSelect := 0;
  elsif navSelect = 1 then
     lightsSelect   := 0;
     socketsSelect  := 1;
     shuttersSelect := 0;
  elsif navSelect = 2 then
     lightsSelect   := 0;
     socketsSelect  := 0;
     shuttersSelect := 1;
  end_if;

  HMI_Index := 4;
  RCU_Index := 3;

  if GetRemoteIPaddress(chanCode := Eth1_uni2, ethAdr := RCU_ethAdr) then
     RCUs_IPs[RCU_Index] := RCU_ethAdr.remoteIP;
  end_if;

  HMIs_Info[HMI_Index].SNo := HMI_Addresses[1];
  HMIs_Info[HMI_Index].readStAdd  := 391;
  HMIs_Info[HMI_Index].writeStAdd := 451;
  HMIs_Info[HMI_Index].readNoPoint  := SIZEOF(HMIs_DataRead[HMI_Index]) / 2;
  HMIs_Info[HMI_Index].writeNoPoint := SIZEOF(HMIs_DataWrite[HMI_Index]) / 2;

  for i := 1 to NumOfHMIsLivingRoom-1 do
    HMIs_Info[HMI_Index+i] := HMIs_Info[HMI_Index];
    HMIs_Info[HMI_Index+i].SNo := HMI_Addresses[i+1];
  end_for;

  afterRestart_TP(IN := IS_COLD_RESTART_PLC or IS_HOT_RESTART_PLC, PT := T#2s );
  afterRestart_TP_FT(CLK := afterRestart_TP.Q);

  if afterRestart_TP_FT.Q then
     SendIamServer := 1;
  end_if;

  controlRoom(RCU_ChCode := ETH1_uni2 , RCU_PingDone := RCUs_PingDone[RCU_Index],
              numOfLights := NumOfLightLivingRoom , numOfOutlets := NumOfOutletLivingRoom , numOfCurtains := NumOfCurtainLivingRoom, numOfMotionSens := NumOfMotionSensLivingRoom,
              lightsOutputDevs := lightsOutputDevs , outletOutputDevs := outletOutputDevs ,
              curtainsUpOutputDevs := curtainsUpOutputDevs , curtainsDwOutputDevs := curtainsDwOutputDevs,
              RCU_CH_IN := void(ETH1_uni2_IN) , LightsStatus := lightsStatusLivingRoom ,OutletsStatus := outletsStatusLivingRoom, MotionSenStatus := motionSensStatus,
              EnLights := EnLights , EnLightsAN := EnLightsAN , EnOutlets := EnOutlets ,EnOutletsAN :=EnOutletsAN ,
              SendIamServer := SendIamServer , GetAllStatus := GetAllStatus);

              //stLightsLivingRoomAN := lightsStatusLivingRoom[1];

  (* FCU[1](enable := enableFCU[1], mode := settingsFCU[1].FCU_Mode, fanSpeed := settingsFCU[1].FCU_FanSpeed, setTemp := setTempFCU_LivingRoom[1], temp := FCU_Temp_LivingRoom, valve := FCU_valve_LivingRoom, fanLow := FCU_fanLow_LivingRoom,
                 fanMed := FCU_fanMed_LivingRoom, fanHigh := FCU_fanHigh_LivingRoom);  *)

   for i := 1 to NumOfLightLivingRoom do
       HMIs_DataWrite[HMI_Index].lightsStatus[i] := BOOL_TO_WORD(lightsStatusLivingRoom[i]);
   end_for;

   for i := 1 to NumOfOutletLivingRoom do
       HMIs_DataWrite[HMI_Index].outletsStatus[i] := BOOL_TO_WORD(outletsStatusLivingRoom[i]);
   end_for;

   for i := 1 to NumOfMotionSensLivingRoom do
       HMIs_DataWrite[HMI_Index].motionSensStatus[i] := BOOL_TO_WORD(motionSensStatus[i]);
   end_for;

  (* for i := 1 to NumOfFCUsLivingRoom do
      HMIs_DataWrite[HMI_Index].FCUs_Status[i] := FCU[i].FCU_Status;
   end_for; *)

   for i := 1 to NumOfHMIsLivingRoom-1 do
     HMIs_DataWrite[HMI_Index+i] := HMIs_DataWrite[HMI_Index];
   end_for;

   for j := 1 to NumOfHMIsLivingRoom do
     for i := 1 to NumOfLightLivingRoom do

         enLights_RT[j,i](CLK := HMIs_DataRead[HMI_Index + j - 1].enLights[i]);

         enLights_FT[j,i](CLK := HMIs_DataRead[HMI_Index + j - 1].enLights[i]);

         if enLights_RT[j,i].Q or enLights_FT[j,i].Q then
            EnLights[i] := 1;
         end_if;
     end_for;
   end_for;

   for j := 1 to NumOfHMIsLivingRoom do
     for i := 1 to NumOfOutletLivingRoom do

         enOutlets_RT[j,i](CLK := HMIs_DataRead[HMI_Index + j - 1].enOutlets[i]);

         enOutlets_FT[j,i](CLK := HMIs_DataRead[HMI_Index + j - 1].enOutlets[i]);

         if enOutlets_RT[j,i].Q or enOutlets_FT[j,i].Q then
            EnOutlets[i] := 1;
         end_if;
     end_for;
   end_for;

   for j := 1 to NumOfHMIsLivingRoom do
     for i := 1 to NumOfCurtainLivingRoom do

         enCurtainsUP_RT[j,i](CLK := HMIs_DataRead[HMI_Index + j - 1].enShutters[i].UP.0);

         enCurtainsUP_FT[j,i](CLK := HMIs_DataRead[HMI_Index + j - 1].enShutters[i].UP.0);

         if enCurtainsUP_RT[j,i].Q or enCurtainsUP_FT[j,i].Q then
            EnCurtainsUp[i] := 1;
         end_if;

         enCurtainsDW_RT[j,i](CLK := HMIs_DataRead[HMI_Index + j - 1].enShutters[i].Dw.0);

         enCurtainsDW_FT[j,i](CLK := HMIs_DataRead[HMI_Index + j - 1].enShutters[i].Dw.0);

         if enCurtainsDW_RT[j,i].Q or enCurtainsDW_FT[j,i].Q then
            EnCurtainsDw[i] := 1;
         end_if;

     end_for;
   end_for;

   (*
   for j := 1 to NumOfHMIsLivingRoom do
      for i := 1 to NumOfFCUsLivingRoom do
          enFCUs_FT[j,i](CLK := HMIs_DataRead[HMI_Index + j - 1].enFCUs[i].onOff);
          enFCUs_RT[j,i](CLK := HMIs_DataRead[HMI_Index + j - 1].enFCUs[i].onOff);

          if enFCUs_FT[j,i].Q then
             enableFCU[i] := 0;
          end_if;
          if enFCUs_RT[j,i].Q then
             enableFCU[i] := 1;
          end_if;

          enFanAuto_RT[j,i](CLK := (HMIs_DataRead[HMI_Index + j - 1].enFCUs[i].fanSpeed = 8));
          enFanLow_RT[j,i](CLK := HMIs_DataRead[HMI_Index + j - 1].enFCUs[i].fanSpeed.0);
          enFanMed_RT[j,i](CLK := HMIs_DataRead[HMI_Index + j - 1].enFCUs[i].fanSpeed.1);
          enFanHigh_RT[j,i](CLK := HMIs_DataRead[HMI_Index + j - 1].enFCUs[i].fanSpeed.2);

          if enFanAuto_RT[j,i].Q then
             settingsFCU[i].FCU_FanSpeed := auto;
          end_if;
          if enFanLow_RT[j,i].Q then
             settingsFCU[i].FCU_FanSpeed := low;
          end_if;
          if enFanMed_RT[j,i].Q then
             settingsFCU[i].FCU_FanSpeed := med;
          end_if;
          if enFanHigh_RT[j,i].Q then
             settingsFCU[i].FCU_FanSpeed := high;
          end_if;

          enFCUCool_RT[j,i](CLK := (HMIs_DataRead[HMI_Index + j - 1].enFCUs[i].mode = 0));
          enFCUFanOnly_RT[j,i](CLK := HMIs_DataRead[HMI_Index + j - 1].enFCUs[i].mode.0);

          if enFCUCool_RT[j,i].Q then
             settingsFCU[i].FCU_Mode := cooling;
          end_if;
          if enFCUFanOnly_RT[j,i].Q then
             settingsFCU[i].FCU_Mode := fanOnly;
          end_if;

          enSetTempIncr_RT[j,i](CLK := HMIs_DataRead[HMI_Index + j - 1].enFCUs[i].SetTempCtrl.0);
          enSetTempIncr_FT[j,i](CLK := HMIs_DataRead[HMI_Index + j - 1].enFCUs[i].SetTempCtrl.0);

          if enSetTempIncr_RT[j,i].Q or enSetTempIncr_FT[j,i].Q then
             setTempFCU_LivingRoom[j] := setTempFCU_LivingRoom[j] + 0.5;
          end_if;

          enSetTempDecr_RT[j,i](CLK := HMIs_DataRead[HMI_Index + j - 1].enFCUs[i].SetTempCtrl.1);
          enSetTempDecr_FT[j,i](CLK := HMIs_DataRead[HMI_Index + j - 1].enFCUs[i].SetTempCtrl.1);

          if enSetTempDecr_RT[j,i].Q or enSetTempDecr_FT[j,i].Q then
             setTempFCU_LivingRoom[j] := setTempFCU_LivingRoom[j] - 0.5;
          end_if;

      end_for;
   end_for; *)

END_PROGRAM

(* ---- PrgMain.ST ---- *)
Var_Global Constant
   numOfRCUS : INT := 7;
End_Var

Var_Global Retain
   RCUs_IPs : Array[1..numOfRCUS] of TIPAdr := [[192,168,0,23],
                                                [192,168,0,15],
                                                [192,168,0,17],
                                                [192,168,0,109],
                                                [192,168,0,110]];
End_Var

Var_Global
   RCUs_PingDone : array[1..numOfRCUS] of BOOL;
End_Var

PROGRAM prgMain
  VAR_INPUT
  END_VAR
  VAR_OUTPUT
  END_VAR
  VAR
  // Check RCUs connection
  ping     : fbPingIP ;
  pingInfo : T_PING_INFO;
  tick     : fbTick;
  pingSwitch : INT;
  IP        : TIPadr;

  //
  currentDT : DT;

  END_VAR

  // check the connection of all RCUs

  tick(IN := 1, PT :=T#1.2s );
  if tick.Q then
     pingSwitch :=  pingSwitch + 1;
  end_if;

  if pingSwitch = numOfRCUS then
     pingSwitch := 0;
  end_if;

  if pingSwitch >= 0 and pingSwitch < numOfRCUS then
     IP := RCUs_IPs[pingSwitch + 1];
  end_if;

  ping(rqPing := tick.Q , hostIP := IP , ttl := 255 , timeLimit :=T#1s ,  pingInfo := pingInfo );

  if pingSwitch >= 0 and pingSwitch < numOfRCUS then
    IF ping.done THEN
       RCUs_PingDone[pingSwitch + 1] :=1;
    END_IF;
    IF ping.busy or ping.err THEN
       RCUs_PingDone[pingSwitch + 1] :=0;
    END_IF;
  end_if;

  currentDT := GetDateTime();

END_PROGRAM

(* ---- PrgMasterRoom.ST ---- *)
VAR_GLOBAL CONSTANT
   NumOfLightMasterRoom      : USINT := 8;
   NumOfOutletMasterRoom     : USINT := 4;
   NumOfCurtainMasterRoom    : USINT := 2;
   NumOfMotionSensMasterRoom : USINT := 1;
   NumOfFCUsMasterRoom       : USINT := 1;
   NumOfHMIsMasterRoom       : USINT := 2;
END_VAR

VAR_GLOBAL RETAIN
   lightsStatusMasterRoom  {PUBLIC_API} : TLightsStatus;
   outletsStatusMasterRoom {PUBLIC_API} : TOutletsStatus;
   setTempFCU_MasterRoom  : Array[1..NumOfFCUsMasterRoom] of REAL := [20];

END_VAR

PROGRAM PrgMasterRoom

  VAR
  //WebMaker
  lightsSelect   : BOOL;
  socketsSelect  : BOOL;
  shuttersSelect : BOOL;
  AC_Select      : BOOL;
  navSelect      : usint;

  //RCU
  RCU_ethAdr   : TRemoteEthAdr;
  RCU_IP : TIPadr := [192, 168, 0, 23];
  RCU_Ch_localPort : UINT;
  Set_IP           : BOOL;
  GetAllStatus  : BOOL;
  SendIamServer : BOOL;

  //controlRoom
  controlRoom   : fbControlRoom ;
  lightsOutputDevs     : TlightsOutputDevs     := [(DevAddress := 1 , loopAddress := 1),(DevAddress := 1 , loopAddress := 2),
                                                   (DevAddress := 1 , loopAddress := 3),(DevAddress := 1 , loopAddress := 4),
                                                   (DevAddress := 1 , loopAddress := 5),(DevAddress := 1 , loopAddress := 6),
                                                   (DevAddress := 1 , loopAddress := 7),(DevAddress := 1 , loopAddress := 8)];

  outletOutputDevs     : ToutletOutputDevs     := [(DevAddress := 1 , loopAddress := 9),(DevAddress := 1 , loopAddress := 10),
                                                   (DevAddress := 2 , loopAddress := 1),(DevAddress := 2 , loopAddress := 2)];

  curtainsUpOutputDevs : TcurtainsUpOutputDevs := [(DevAddress := 2 , loopAddress := 3),(DevAddress := 2 , loopAddress := 5)];
  curtainsDwOutputDevs : TcurtainsDwOutputDevs := [(DevAddress := 2 , loopAddress := 4),(DevAddress := 2 , loopAddress := 6)];

  motionSensOutputDevs : TMotionSensOutputDevs := [(DevAddress := 1 , loopAddress := 1)];

  EnLights                            : TEnLights     ;
  EnLightsAN       {PUBLIC_API}       : TEnLightsAN   ;
  EnOutlets                           : TEnOutlets    ;
  EnOutletsAN      {PUBLIC_API}       : TEnOutletsAN  ;
  EnCurtainsUp     {PUBLIC_API}       : TEnCurtainsUp ;
  EnCurtainsDw     {PUBLIC_API}       : TEnCurtainsDW ;
   //EnLightsMasterRoomAN1  {PUBLIC_API}      : TEnLightsAN1    ;
   //stLightsMasterRoomAN  {PUBLIC_API}       : BOOL     ;
  //curtainsFB       : TCurtainsFB;
  //CurtainPositWm   : TCurtainPositWm;

  //
  enLights_RT  : Array[1..NumOfHMIsMasterRoom,1..NumOfLightMasterRoom] of R_TRIG;
  enLights_FT  : Array[1..NumOfHMIsMasterRoom,1..NumOfLightMasterRoom] of F_TRIG;

  enOutlets_RT : Array[1..NumOfHMIsMasterRoom,1..NumOfOutletMasterRoom] of R_TRIG;
  enOutlets_FT : Array[1..NumOfHMIsMasterRoom,1..NumOfOutletMasterRoom] of F_TRIG;

  enCurtainsUP_RT : Array[1..NumOfHMIsMasterRoom,1..NumOfCurtainMasterRoom] of R_TRIG;
  enCurtainsUP_FT : Array[1..NumOfHMIsMasterRoom,1..NumOfCurtainMasterRoom] of F_TRIG;

  enCurtainsDW_RT : Array[1..NumOfHMIsMasterRoom,1..NumOfCurtainMasterRoom] of R_TRIG;
  enCurtainsDW_FT : Array[1..NumOfHMIsMasterRoom,1..NumOfCurtainMasterRoom] of F_TRIG;

  //
  i , j : USINT;
  afterRestart_TP : TP;
  afterRestart_TP_FT : F_TRIG;

  //
  motionSensStatus                : TMotionSensStatus;
  CurtainsUpStatus   {PUBLIC_API} : TCurtainsUpStatus;
  CurtainsDwStatus   {PUBLIC_API} : TCurtainsDwStatus;

  // FCU VARS
  FCU          : Array[1..NumOfFCUsMasterRoom] of fbControlFCU;
  enableFCU    : Array[1..NumOfFCUsMasterRoom] of BOOL;
  settingsFCU  : Array[1..NumOfFCUsMasterRoom] of TFCU_Settings;

  //modeFCU      : Array[1..NumOfFCUsMasterRoom] of TFCU_Mode;
  //fanSpeedFCU  : Array[1..NumOfFCUsMasterRoom] of TFCU_FanSpeed;

  enFCUs_FT    : Array[1..NumOfHMIsMasterRoom,1..NumOfFCUsMasterRoom] of F_TRIG;
  enFCUs_RT    : Array[1..NumOfHMIsMasterRoom,1..NumOfFCUsMasterRoom] of R_TRIG;

  enFanHigh_RT : Array[1..NumOfHMIsMasterRoom,1..NumOfFCUsMasterRoom] of R_TRIG;
  enFanMed_RT  : Array[1..NumOfHMIsMasterRoom,1..NumOfFCUsMasterRoom] of R_TRIG;
  enFanLow_RT  : Array[1..NumOfHMIsMasterRoom,1..NumOfFCUsMasterRoom] of R_TRIG;
  enFanAuto_RT : Array[1..NumOfHMIsMasterRoom,1..NumOfFCUsMasterRoom] of R_TRIG;

  enFCUCool_RT    : Array[1..NumOfHMIsMasterRoom,1..NumOfFCUsMasterRoom] of R_TRIG;
  enFCUFanOnly_RT : Array[1..NumOfHMIsMasterRoom,1..NumOfFCUsMasterRoom] of R_TRIG;

  enSetTempIncr_RT : Array[1..NumOfHMIsMasterRoom,1..NumOfFCUsMasterRoom] of R_TRIG;
  enSetTempIncr_FT : Array[1..NumOfHMIsMasterRoom,1..NumOfFCUsMasterRoom] of F_TRIG;

  enSetTempDecr_RT : Array[1..NumOfHMIsMasterRoom,1..NumOfFCUsMasterRoom] of R_TRIG;
  enSetTempDecr_FT : Array[1..NumOfHMIsMasterRoom,1..NumOfFCUsMasterRoom] of F_TRIG;

  //HMIs[1..num
  HMI_Index : USINT;
  RCU_Index : USINT;
  HMI_Addresses : Array[1..NumOfHMIsMasterRoom] of USINT := [4, 6];

  END_VAR

   if navSelect = 0 then
     lightsSelect   := 1;
     socketsSelect  := 0;
     shuttersSelect := 0;
     AC_Select      := 0;
  elsif navSelect = 1 then
     lightsSelect   := 0;
     socketsSelect  := 1;
     shuttersSelect := 0;
     AC_Select      := 0;
  elsif navSelect = 2 then
     lightsSelect   := 0;
     socketsSelect  := 0;
     shuttersSelect := 1;
     AC_Select      := 0;
  elsif navSelect = 3 then
     lightsSelect   := 0;
     socketsSelect  := 0;
     shuttersSelect := 0;
     AC_Select      := 1;
  end_if;

  HMI_Index := 8;
  RCU_Index := 6;

  if GetRemoteIPaddress(chanCode := Eth1_uni5, ethAdr := RCU_ethAdr) then
     RCUs_IPs[RCU_Index] := RCU_ethAdr.remoteIP;
  end_if;

  HMIs_Info[HMI_Index].SNo := HMI_Addresses[1];
  HMIs_Info[HMI_Index].readStAdd  := 781;
  HMIs_Info[HMI_Index].writeStAdd := 841;
  HMIs_Info[HMI_Index].readNoPoint  := SIZEOF(HMIs_DataRead[HMI_Index]) / 2;
  HMIs_Info[HMI_Index].writeNoPoint := SIZEOF(HMIs_DataWrite[HMI_Index]) / 2;

  for i := 1 to NumOfHMIsMasterRoom-1 do
    HMIs_Info[HMI_Index+i] := HMIs_Info[HMI_Index];
    HMIs_Info[HMI_Index+i].SNo := HMI_Addresses[i+1];
  end_for;

  afterRestart_TP(IN := IS_COLD_RESTART_PLC or IS_HOT_RESTART_PLC, PT := T#2s );
  afterRestart_TP_FT(CLK := afterRestart_TP.Q);

  if afterRestart_TP_FT.Q then
     SendIamServer := 1;
  end_if;

  controlRoom(RCU_ChCode := ETH1_uni5 , RCU_PingDone := RCUs_PingDone[RCU_Index],
              numOfLights := NumOfLightMasterRoom , numOfOutlets := NumOfOutletMasterRoom , numOfCurtains := NumOfCurtainMasterRoom, numOfMotionSens := NumOfMotionSensMasterRoom,
              lightsOutputDevs := lightsOutputDevs , outletOutputDevs := outletOutputDevs ,
              curtainsUpOutputDevs := curtainsUpOutputDevs , curtainsDwOutputDevs := curtainsDwOutputDevs,
              RCU_CH_IN := void(ETH1_uni5_IN) , LightsStatus := lightsStatusMasterRoom ,OutletsStatus := outletsStatusMasterRoom, MotionSenStatus := motionSensStatus,
              EnLights := EnLights , EnLightsAN := EnLightsAN , EnOutlets := EnOutlets ,EnOutletsAN :=EnOutletsAN ,
              SendIamServer := SendIamServer , GetAllStatus := GetAllStatus);

              //stLightsMasterRoomAN := lightsStatusMasterRoom[1];

   FCU[1](enable := enableFCU[1], mode := settingsFCU[1].FCU_Mode, fanSpeed := settingsFCU[1].FCU_FanSpeed, setTemp := setTempFCU_MasterRoom[1], temp := FCU_Temp_MasterRoom, valve := FCU_valve_MasterRoom, fanLow := FCU_fanLow_MasterRoom,
                 fanMed := FCU_fanMed_MasterRoom, fanHigh := FCU_fanHigh_MasterRoom);

   for i := 1 to NumOfLightMasterRoom do
       HMIs_DataWrite[HMI_Index].lightsStatus[i] := BOOL_TO_WORD(lightsStatusMasterRoom[i]);
   end_for;

   for i := 1 to NumOfOutletMasterRoom do
       HMIs_DataWrite[HMI_Index].outletsStatus[i] := BOOL_TO_WORD(outletsStatusMasterRoom[i]);
   end_for;

   for i := 1 to NumOfMotionSensMasterRoom do
       HMIs_DataWrite[HMI_Index].motionSensStatus[i] := BOOL_TO_WORD(motionSensStatus[i]);
   end_for;

   for i := 1 to NumOfFCUsMasterRoom do
      HMIs_DataWrite[HMI_Index].FCUs_Status[i] := FCU[i].FCU_Status;
   end_for;

   for i := 1 to NumOfHMIsMasterRoom-1 do
     HMIs_DataWrite[HMI_Index+i] := HMIs_DataWrite[HMI_Index];
   end_for;

   for j := 1 to NumOfHMIsMasterRoom do
     for i := 1 to NumOfLightMasterRoom do

         enLights_RT[j,i](CLK := HMIs_DataRead[HMI_Index + j - 1].enLights[i]);

         enLights_FT[j,i](CLK := HMIs_DataRead[HMI_Index + j - 1].enLights[i]);

         if enLights_RT[j,i].Q or enLights_FT[j,i].Q then
            EnLights[i] := 1;
         end_if;
     end_for;
   end_for;

   for j := 1 to NumOfHMIsMasterRoom do
     for i := 1 to NumOfOutletMasterRoom do

         enOutlets_RT[j,i](CLK := HMIs_DataRead[HMI_Index + j - 1].enOutlets[i]);

         enOutlets_FT[j,i](CLK := HMIs_DataRead[HMI_Index + j - 1].enOutlets[i]);

         if enOutlets_RT[j,i].Q or enOutlets_FT[j,i].Q then
            EnOutlets[i] := 1;
         end_if;
     end_for;
   end_for;

   for j := 1 to NumOfHMIsMasterRoom do
     for i := 1 to NumOfCurtainMasterRoom do

         enCurtainsUP_RT[j,i](CLK := HMIs_DataRead[HMI_Index + j - 1].enShutters[i].UP.0);

         enCurtainsUP_FT[j,i](CLK := HMIs_DataRead[HMI_Index + j - 1].enShutters[i].UP.0);

         if enCurtainsUP_RT[j,i].Q or enCurtainsUP_FT[j,i].Q then
            EnCurtainsUp[i] := 1;
         end_if;

         enCurtainsDW_RT[j,i](CLK := HMIs_DataRead[HMI_Index + j - 1].enShutters[i].Dw.0);

         enCurtainsDW_FT[j,i](CLK := HMIs_DataRead[HMI_Index + j - 1].enShutters[i].Dw.0);

         if enCurtainsDW_RT[j,i].Q or enCurtainsDW_FT[j,i].Q then
            EnCurtainsDw[i] := 1;
         end_if;

     end_for;
   end_for;

   for j := 1 to NumOfHMIsMasterRoom do
      for i := 1 to NumOfFCUsMasterRoom do
          enFCUs_FT[j,i](CLK := HMIs_DataRead[HMI_Index + j - 1].enFCUs[i].onOff);
          enFCUs_RT[j,i](CLK := HMIs_DataRead[HMI_Index + j - 1].enFCUs[i].onOff);

          if enFCUs_FT[j,i].Q then
             enableFCU[i] := 0;
          end_if;
          if enFCUs_RT[j,i].Q then
             enableFCU[i] := 1;
          end_if;

          enFanAuto_RT[j,i](CLK := (HMIs_DataRead[HMI_Index + j - 1].enFCUs[i].fanSpeed = 8));
          enFanLow_RT[j,i](CLK := HMIs_DataRead[HMI_Index + j - 1].enFCUs[i].fanSpeed.0);
          enFanMed_RT[j,i](CLK := HMIs_DataRead[HMI_Index + j - 1].enFCUs[i].fanSpeed.1);
          enFanHigh_RT[j,i](CLK := HMIs_DataRead[HMI_Index + j - 1].enFCUs[i].fanSpeed.2);

          if enFanAuto_RT[j,i].Q then
             settingsFCU[i].FCU_FanSpeed := auto;
          end_if;
          if enFanLow_RT[j,i].Q then
             settingsFCU[i].FCU_FanSpeed := low;
          end_if;
          if enFanMed_RT[j,i].Q then
             settingsFCU[i].FCU_FanSpeed := med;
          end_if;
          if enFanHigh_RT[j,i].Q then
             settingsFCU[i].FCU_FanSpeed := high;
          end_if;

          enFCUCool_RT[j,i](CLK := (HMIs_DataRead[HMI_Index + j - 1].enFCUs[i].mode = 0));
          enFCUFanOnly_RT[j,i](CLK := HMIs_DataRead[HMI_Index + j - 1].enFCUs[i].mode.0);

          if enFCUCool_RT[j,i].Q then
             settingsFCU[i].FCU_Mode := cooling;
          end_if;
          if enFCUFanOnly_RT[j,i].Q then
             settingsFCU[i].FCU_Mode := fanOnly;
          end_if;

          enSetTempIncr_RT[j,i](CLK := HMIs_DataRead[HMI_Index + j - 1].enFCUs[i].SetTempCtrl.0);
          enSetTempIncr_FT[j,i](CLK := HMIs_DataRead[HMI_Index + j - 1].enFCUs[i].SetTempCtrl.0);

          if enSetTempIncr_RT[j,i].Q or enSetTempIncr_FT[j,i].Q then
             setTempFCU_MasterRoom[j] := setTempFCU_MasterRoom[j] + 0.5;
          end_if;

          enSetTempDecr_RT[j,i](CLK := HMIs_DataRead[HMI_Index + j - 1].enFCUs[i].SetTempCtrl.1);
          enSetTempDecr_FT[j,i](CLK := HMIs_DataRead[HMI_Index + j - 1].enFCUs[i].SetTempCtrl.1);

          if enSetTempDecr_RT[j,i].Q or enSetTempDecr_FT[j,i].Q then
             setTempFCU_MasterRoom[j] := setTempFCU_MasterRoom[j] - 0.5;
          end_if;

      end_for;
   end_for;

END_PROGRAM

(* ---- PrgRoom4.ST ---- *)
VAR_GLOBAL CONSTANT
   NumOfLightRoom4      : USINT := 6;
   NumOfOutletRoom4     : USINT := 2;
   NumOfCurtainRoom4    : USINT := 1;
   NumOfMotionSensRoom4 : USINT := 2;
   NumOfFCUsRoom4       : USINT := 1;
   NumOfHMIsRoom4       : USINT := 2;
END_VAR

VAR_GLOBAL RETAIN
   lightsStatusRoom4  {PUBLIC_API} : TLightsStatus;
   outletsStatusRoom4 {PUBLIC_API} : TOutletsStatus;
   setTempFCU_Room4  : Array[1..NumOfFCUsRoom4] of REAL := [20];

END_VAR

PROGRAM PrgRoom4

  VAR
  //WebMaker
  lightsSelect   : BOOL;
  socketsSelect  : BOOL;
  shuttersSelect : BOOL;
  AC_Select      : BOOL;
  navSelect      : usint;

  //RCU
  RCU_ethAdr   : TRemoteEthAdr;
  RCU_IP : TIPadr := [192, 168, 0, 23];
  RCU_Ch_localPort : UINT;
  Set_IP           : BOOL;
  GetAllStatus  : BOOL;
  SendIamServer : BOOL;

  //controlRoom
  controlRoom   : fbControlRoom ;
  lightsOutputDevs     : TlightsOutputDevs     := [(DevAddress := 1 , loopAddress := 1),(DevAddress := 1 , loopAddress := 2),
                                                   (DevAddress := 1 , loopAddress := 3),(DevAddress := 1 , loopAddress := 4),
                                                   (DevAddress := 1 , loopAddress := 5),(DevAddress := 1 , loopAddress := 6)];

  outletOutputDevs     : ToutletOutputDevs     := [(DevAddress := 1 , loopAddress := 7),(DevAddress := 1 , loopAddress := 8)];

  curtainsUpOutputDevs : TcurtainsUpOutputDevs := [(DevAddress := 1 , loopAddress := 9)];
  curtainsDwOutputDevs : TcurtainsDwOutputDevs := [(DevAddress := 1 , loopAddress := 10)];

  motionSensOutputDevs : TMotionSensOutputDevs := [(DevAddress := 1 , loopAddress := 1),(DevAddress := 1 , loopAddress := 2)];

  EnLights                            : TEnLights     ;
  EnLightsAN       {PUBLIC_API}       : TEnLightsAN   ;
  EnOutlets                           : TEnOutlets    ;
  EnOutletsAN      {PUBLIC_API}       : TEnOutletsAN  ;
  EnCurtainsUp     {PUBLIC_API}       : TEnCurtainsUp ;
  EnCurtainsDw     {PUBLIC_API}       : TEnCurtainsDW ;
   //EnLightsRoom4AN1  {PUBLIC_API}      : TEnLightsAN1    ;
   //stLightsRoom4AN  {PUBLIC_API}       : BOOL     ;
  //curtainsFB       : TCurtainsFB;
  //CurtainPositWm   : TCurtainPositWm;

  //
  enLights_RT  : Array[1..NumOfHMIsRoom4,1..NumOfLightRoom4] of R_TRIG;
  enLights_FT  : Array[1..NumOfHMIsRoom4,1..NumOfLightRoom4] of F_TRIG;

  enOutlets_RT : Array[1..NumOfHMIsRoom4,1..NumOfOutletRoom4] of R_TRIG;
  enOutlets_FT : Array[1..NumOfHMIsRoom4,1..NumOfOutletRoom4] of F_TRIG;

  enCurtainsUP_RT : Array[1..NumOfHMIsRoom4,1..NumOfCurtainRoom4] of R_TRIG;
  enCurtainsUP_FT : Array[1..NumOfHMIsRoom4,1..NumOfCurtainRoom4] of F_TRIG;

  enCurtainsDW_RT : Array[1..NumOfHMIsRoom4,1..NumOfCurtainRoom4] of R_TRIG;
  enCurtainsDW_FT : Array[1..NumOfHMIsRoom4,1..NumOfCurtainRoom4] of F_TRIG;

  //
  i , j : USINT;
  afterRestart_TP : TP;
  afterRestart_TP_FT : F_TRIG;

  //
  motionSensStatus                : TMotionSensStatus;
  CurtainsUpStatus   {PUBLIC_API} : TCurtainsUpStatus;
  CurtainsDwStatus   {PUBLIC_API} : TCurtainsDwStatus;

  // FCU VARS
  FCU          : Array[1..NumOfFCUsRoom4] of fbControlFCU;
  enableFCU    : Array[1..NumOfFCUsRoom4] of BOOL;
  settingsFCU  : Array[1..NumOfFCUsRoom4] of TFCU_Settings;

  //modeFCU      : Array[1..NumOfFCUsRoom4] of TFCU_Mode;
  //fanSpeedFCU  : Array[1..NumOfFCUsRoom4] of TFCU_FanSpeed;

  enFCUs_FT    : Array[1..NumOfHMIsRoom4,1..NumOfFCUsRoom4] of F_TRIG;
  enFCUs_RT    : Array[1..NumOfHMIsRoom4,1..NumOfFCUsRoom4] of R_TRIG;

  enFanHigh_RT : Array[1..NumOfHMIsRoom4,1..NumOfFCUsRoom4] of R_TRIG;
  enFanMed_RT  : Array[1..NumOfHMIsRoom4,1..NumOfFCUsRoom4] of R_TRIG;
  enFanLow_RT  : Array[1..NumOfHMIsRoom4,1..NumOfFCUsRoom4] of R_TRIG;
  enFanAuto_RT : Array[1..NumOfHMIsRoom4,1..NumOfFCUsRoom4] of R_TRIG;

  enFCUCool_RT    : Array[1..NumOfHMIsRoom4,1..NumOfFCUsRoom4] of R_TRIG;
  enFCUFanOnly_RT : Array[1..NumOfHMIsRoom4,1..NumOfFCUsRoom4] of R_TRIG;

  enSetTempIncr_RT : Array[1..NumOfHMIsRoom4,1..NumOfFCUsRoom4] of R_TRIG;
  enSetTempIncr_FT : Array[1..NumOfHMIsRoom4,1..NumOfFCUsRoom4] of F_TRIG;

  enSetTempDecr_RT : Array[1..NumOfHMIsRoom4,1..NumOfFCUsRoom4] of R_TRIG;
  enSetTempDecr_FT : Array[1..NumOfHMIsRoom4,1..NumOfFCUsRoom4] of F_TRIG;

  //HMIs[1..num
  HMI_Index : USINT;
  RCU_Index : USINT;
  HMI_Addresses : Array[1..NumOfHMIsRoom4] of USINT := [9, 11];

  END_VAR

   if navSelect = 0 then
     lightsSelect   := 1;
     socketsSelect  := 0;
     shuttersSelect := 0;
     AC_Select      := 0;
  elsif navSelect = 1 then
     lightsSelect   := 0;
     socketsSelect  := 1;
     shuttersSelect := 0;
     AC_Select      := 0;
  elsif navSelect = 2 then
     lightsSelect   := 0;
     socketsSelect  := 0;
     shuttersSelect := 1;
     AC_Select      := 0;
  elsif navSelect = 3 then
     lightsSelect   := 0;
     socketsSelect  := 0;
     shuttersSelect := 0;
     AC_Select      := 1;
  end_if;

  HMI_Index := 10;
  RCU_Index := 7;

  if GetRemoteIPaddress(chanCode := Eth1_uni6, ethAdr := RCU_ethAdr) then
     RCUs_IPs[RCU_Index] := RCU_ethAdr.remoteIP;
  end_if;

  HMIs_Info[HMI_Index].SNo := HMI_Addresses[1];
  HMIs_Info[HMI_Index].readStAdd  := 1301;
  HMIs_Info[HMI_Index].writeStAdd := 1361;
  HMIs_Info[HMI_Index].readNoPoint  := SIZEOF(HMIs_DataRead[HMI_Index]) / 2;
  HMIs_Info[HMI_Index].writeNoPoint := SIZEOF(HMIs_DataWrite[HMI_Index]) / 2;

  for i := 1 to NumOfHMIsRoom4-1 do
    HMIs_Info[HMI_Index+i] := HMIs_Info[HMI_Index];
    HMIs_Info[HMI_Index+i].SNo := HMI_Addresses[i+1];
  end_for;

  afterRestart_TP(IN := IS_COLD_RESTART_PLC or IS_HOT_RESTART_PLC, PT := T#2s );
  afterRestart_TP_FT(CLK := afterRestart_TP.Q);

  if afterRestart_TP_FT.Q then
     SendIamServer := 1;
  end_if;

  controlRoom(RCU_ChCode := ETH1_uni6 , RCU_PingDone := RCUs_PingDone[RCU_Index],
              numOfLights := NumOfLightRoom4 , numOfOutlets := NumOfOutletRoom4 , numOfCurtains := NumOfCurtainRoom4, numOfMotionSens := NumOfMotionSensRoom4,
              lightsOutputDevs := lightsOutputDevs , outletOutputDevs := outletOutputDevs ,
              curtainsUpOutputDevs := curtainsUpOutputDevs , curtainsDwOutputDevs := curtainsDwOutputDevs,
              RCU_CH_IN := void(ETH1_uni6_IN) , LightsStatus := lightsStatusRoom4 ,OutletsStatus := outletsStatusRoom4, MotionSenStatus := motionSensStatus,
              EnLights := EnLights , EnLightsAN := EnLightsAN , EnOutlets := EnOutlets ,EnOutletsAN :=EnOutletsAN ,
              SendIamServer := SendIamServer , GetAllStatus := GetAllStatus);

              //stLightsRoom4AN := lightsStatusRoom4[1];

   FCU[1](enable := enableFCU[1], mode := settingsFCU[1].FCU_Mode, fanSpeed := settingsFCU[1].FCU_FanSpeed, setTemp := setTempFCU_Room4[1], temp := FCU_Temp_Room4, valve := FCU_valve_Room4, fanLow := FCU_fanLow_Room4,
                 fanMed := FCU_fanMed_Room4, fanHigh := FCU_fanHigh_Room4);

   for i := 1 to NumOfLightRoom4 do
       HMIs_DataWrite[HMI_Index].lightsStatus[i] := BOOL_TO_WORD(lightsStatusRoom4[i]);
   end_for;

   for i := 1 to NumOfOutletRoom4 do
       HMIs_DataWrite[HMI_Index].outletsStatus[i] := BOOL_TO_WORD(outletsStatusRoom4[i]);
   end_for;

   for i := 1 to NumOfMotionSensRoom4 do
       HMIs_DataWrite[HMI_Index].motionSensStatus[i] := BOOL_TO_WORD(motionSensStatus[i]);
   end_for;

   for i := 1 to NumOfFCUsRoom4 do
      HMIs_DataWrite[HMI_Index].FCUs_Status[i] := FCU[i].FCU_Status;
   end_for;

   for i := 1 to NumOfHMIsRoom4-1 do
     HMIs_DataWrite[HMI_Index+i] := HMIs_DataWrite[HMI_Index];
   end_for;

   for j := 1 to NumOfHMIsRoom4 do
     for i := 1 to NumOfLightRoom4 do

         enLights_RT[j,i](CLK := HMIs_DataRead[HMI_Index + j - 1].enLights[i]);

         enLights_FT[j,i](CLK := HMIs_DataRead[HMI_Index + j - 1].enLights[i]);

         if enLights_RT[j,i].Q or enLights_FT[j,i].Q then
            EnLights[i] := 1;
         end_if;
     end_for;
   end_for;

   for j := 1 to NumOfHMIsRoom4 do
     for i := 1 to NumOfOutletRoom4 do

         enOutlets_RT[j,i](CLK := HMIs_DataRead[HMI_Index + j - 1].enOutlets[i]);

         enOutlets_FT[j,i](CLK := HMIs_DataRead[HMI_Index + j - 1].enOutlets[i]);

         if enOutlets_RT[j,i].Q or enOutlets_FT[j,i].Q then
            EnOutlets[i] := 1;
         end_if;
     end_for;
   end_for;

   for j := 1 to NumOfHMIsRoom4 do
     for i := 1 to NumOfCurtainRoom4 do

         enCurtainsUP_RT[j,i](CLK := HMIs_DataRead[HMI_Index + j - 1].enShutters[i].UP.0);

         enCurtainsUP_FT[j,i](CLK := HMIs_DataRead[HMI_Index + j - 1].enShutters[i].UP.0);

         if enCurtainsUP_RT[j,i].Q or enCurtainsUP_FT[j,i].Q then
            EnCurtainsUp[i] := 1;
         end_if;

         enCurtainsDW_RT[j,i](CLK := HMIs_DataRead[HMI_Index + j - 1].enShutters[i].Dw.0);

         enCurtainsDW_FT[j,i](CLK := HMIs_DataRead[HMI_Index + j - 1].enShutters[i].Dw.0);

         if enCurtainsDW_RT[j,i].Q or enCurtainsDW_FT[j,i].Q then
            EnCurtainsDw[i] := 1;
         end_if;

     end_for;
   end_for;

   for j := 1 to NumOfHMIsRoom4 do
      for i := 1 to NumOfFCUsRoom4 do
          enFCUs_FT[j,i](CLK := HMIs_DataRead[HMI_Index + j - 1].enFCUs[i].onOff);
          enFCUs_RT[j,i](CLK := HMIs_DataRead[HMI_Index + j - 1].enFCUs[i].onOff);

          if enFCUs_FT[j,i].Q then
             enableFCU[i] := 0;
          end_if;
          if enFCUs_RT[j,i].Q then
             enableFCU[i] := 1;
          end_if;

          enFanAuto_RT[j,i](CLK := (HMIs_DataRead[HMI_Index + j - 1].enFCUs[i].fanSpeed = 8));
          enFanLow_RT[j,i](CLK := HMIs_DataRead[HMI_Index + j - 1].enFCUs[i].fanSpeed.0);
          enFanMed_RT[j,i](CLK := HMIs_DataRead[HMI_Index + j - 1].enFCUs[i].fanSpeed.1);
          enFanHigh_RT[j,i](CLK := HMIs_DataRead[HMI_Index + j - 1].enFCUs[i].fanSpeed.2);

          if enFanAuto_RT[j,i].Q then
             settingsFCU[i].FCU_FanSpeed := auto;
          end_if;
          if enFanLow_RT[j,i].Q then
             settingsFCU[i].FCU_FanSpeed := low;
          end_if;
          if enFanMed_RT[j,i].Q then
             settingsFCU[i].FCU_FanSpeed := med;
          end_if;
          if enFanHigh_RT[j,i].Q then
             settingsFCU[i].FCU_FanSpeed := high;
          end_if;

          enFCUCool_RT[j,i](CLK := (HMIs_DataRead[HMI_Index + j - 1].enFCUs[i].mode = 0));
          enFCUFanOnly_RT[j,i](CLK := HMIs_DataRead[HMI_Index + j - 1].enFCUs[i].mode.0);

          if enFCUCool_RT[j,i].Q then
             settingsFCU[i].FCU_Mode := cooling;
          end_if;
          if enFCUFanOnly_RT[j,i].Q then
             settingsFCU[i].FCU_Mode := fanOnly;
          end_if;

          enSetTempIncr_RT[j,i](CLK := HMIs_DataRead[HMI_Index + j - 1].enFCUs[i].SetTempCtrl.0);
          enSetTempIncr_FT[j,i](CLK := HMIs_DataRead[HMI_Index + j - 1].enFCUs[i].SetTempCtrl.0);

          if enSetTempIncr_RT[j,i].Q or enSetTempIncr_FT[j,i].Q then
             setTempFCU_Room4[j] := setTempFCU_Room4[j] + 0.5;
          end_if;

          enSetTempDecr_RT[j,i](CLK := HMIs_DataRead[HMI_Index + j - 1].enFCUs[i].SetTempCtrl.1);
          enSetTempDecr_FT[j,i](CLK := HMIs_DataRead[HMI_Index + j - 1].enFCUs[i].SetTempCtrl.1);

          if enSetTempDecr_RT[j,i].Q or enSetTempDecr_FT[j,i].Q then
             setTempFCU_Room4[j] := setTempFCU_Room4[j] - 0.5;
          end_if;

      end_for;
   end_for;

END_PROGRAM

(* ---- PrgServiceRoom.ST ---- *)
VAR_GLOBAL CONSTANT
   NumOfLightServiceRoom      : USINT := 3;
   NumOfOutletServiceRoom     : USINT := 5;
   NumOfCurtainServiceRoom    : USINT := 0;
   NumOfMotionSensServiceRoom : USINT := 1;
   NumOfFCUsServiceRoom       : USINT := 0;
   NumOfHMIsServiceRoom       : USINT := 1;
END_VAR

VAR_GLOBAL RETAIN
   lightsStatusServiceRoom  {PUBLIC_API} : TLightsStatus;
   outletsStatusServiceRoom {PUBLIC_API} : TOutletsStatus;
 (*  setTempFCU_ServiceRoom  : Array[1..NumOfFCUsServiceRoom] of REAL := [20];
   *)

END_VAR

PROGRAM PrgServiceRoom

  VAR
  //WebMaker
  lightsSelect   : BOOL;
  socketsSelect  : BOOL;
  shuttersSelect : BOOL;
  AC_Select      : BOOL;
  navSelect      : usint;

  //RCU
  RCU_ethAdr   : TRemoteEthAdr;
  RCU_IP : TIPadr := [192, 168, 0, 23];
  RCU_Ch_localPort : UINT;
  Set_IP           : BOOL;
  GetAllStatus  : BOOL;
  SendIamServer : BOOL;

  //controlRoom
  controlRoom   : fbControlRoom ;
  lightsOutputDevs     : TlightsOutputDevs     := [(DevAddress := 1 , loopAddress := 1),(DevAddress := 1 , loopAddress := 2),
                                                   (DevAddress := 1 , loopAddress := 3)];

  outletOutputDevs     : ToutletOutputDevs     := [(DevAddress := 1 , loopAddress := 4),(DevAddress := 1 , loopAddress := 5),
                                                   (DevAddress := 1 , loopAddress := 6),(DevAddress := 1 , loopAddress := 7), (DevAddress := 1 , loopAddress := 8)];

  (*curtainsUpOutputDevs : TcurtainsUpOutputDevs := [(DevAddress := 1 , loopAddress := 8)];
  curtainsDwOutputDevs : TcurtainsDwOutputDevs := [(DevAddress := 1 , loopAddress := 9)];*)

  motionSensOutputDevs : TMotionSensOutputDevs := [(DevAddress := 1 , loopAddress := 1)];

  EnLights                            : TEnLights     ;
  EnLightsAN       {PUBLIC_API}       : TEnLightsAN   ;
  EnOutlets                           : TEnOutlets    ;
  EnOutletsAN      {PUBLIC_API}       : TEnOutletsAN  ;
  EnCurtainsUp     {PUBLIC_API}       : TEnCurtainsUp ;
  EnCurtainsDw     {PUBLIC_API}       : TEnCurtainsDW ;
   //EnLightsServiceRoomAN1  {PUBLIC_API}      : TEnLightsAN1    ;
   //stLightsServiceRoomAN  {PUBLIC_API}       : BOOL     ;
  //curtainsFB       : TCurtainsFB;
  //CurtainPositWm   : TCurtainPositWm;

  //
  enLights_RT  : Array[1..NumOfHMIsServiceRoom,1..NumOfLightServiceRoom] of R_TRIG;
  enLights_FT  : Array[1..NumOfHMIsServiceRoom,1..NumOfLightServiceRoom] of F_TRIG;

  enOutlets_RT : Array[1..NumOfHMIsServiceRoom,1..NumOfOutletServiceRoom] of R_TRIG;
  enOutlets_FT : Array[1..NumOfHMIsServiceRoom,1..NumOfOutletServiceRoom] of F_TRIG;
  (*
  enCurtainsUP_RT : Array[1..NumOfHMIsServiceRoom,1..NumOfCurtainServiceRoom] of R_TRIG;
  enCurtainsUP_FT : Array[1..NumOfHMIsServiceRoom,1..NumOfCurtainServiceRoom] of F_TRIG;

  enCurtainsDW_RT : Array[1..NumOfHMIsServiceRoom,1..NumOfCurtainServiceRoom] of R_TRIG;
  enCurtainsDW_FT : Array[1..NumOfHMIsServiceRoom,1..NumOfCurtainServiceRoom] of F_TRIG; *)

  //
  i , j : USINT;
  afterRestart_TP : TP;
  afterRestart_TP_FT : F_TRIG;

  //
  motionSensStatus                : TMotionSensStatus;
  CurtainsUpStatus   {PUBLIC_API} : TCurtainsUpStatus;
  CurtainsDwStatus   {PUBLIC_API} : TCurtainsDwStatus;

  // FCU VARS
  (*FCU          : Array[1..NumOfFCUsServiceRoom] of fbControlFCU;
  enableFCU    : Array[1..NumOfFCUsServiceRoom] of BOOL;
  settingsFCU  : Array[1..NumOfFCUsServiceRoom] of TFCU_Settings;

  //modeFCU      : Array[1..NumOfFCUsServiceRoom] of TFCU_Mode;
  //fanSpeedFCU  : Array[1..NumOfFCUsServiceRoom] of TFCU_FanSpeed;

  enFCUs_FT    : Array[1..NumOfHMIsServiceRoom,1..NumOfFCUsServiceRoom] of F_TRIG;
  enFCUs_RT    : Array[1..NumOfHMIsServiceRoom,1..NumOfFCUsServiceRoom] of R_TRIG;

  enFanHigh_RT : Array[1..NumOfHMIsServiceRoom,1..NumOfFCUsServiceRoom] of R_TRIG;
  enFanMed_RT  : Array[1..NumOfHMIsServiceRoom,1..NumOfFCUsServiceRoom] of R_TRIG;
  enFanLow_RT  : Array[1..NumOfHMIsServiceRoom,1..NumOfFCUsServiceRoom] of R_TRIG;
  enFanAuto_RT : Array[1..NumOfHMIsServiceRoom,1..NumOfFCUsServiceRoom] of R_TRIG;

  enFCUCool_RT    : Array[1..NumOfHMIsServiceRoom,1..NumOfFCUsServiceRoom] of R_TRIG;
  enFCUFanOnly_RT : Array[1..NumOfHMIsServiceRoom,1..NumOfFCUsServiceRoom] of R_TRIG;

  enSetTempIncr_RT : Array[1..NumOfHMIsServiceRoom,1..NumOfFCUsServiceRoom] of R_TRIG;
  enSetTempIncr_FT : Array[1..NumOfHMIsServiceRoom,1..NumOfFCUsServiceRoom] of F_TRIG;

  enSetTempDecr_RT : Array[1..NumOfHMIsServiceRoom,1..NumOfFCUsServiceRoom] of R_TRIG;
  enSetTempDecr_FT : Array[1..NumOfHMIsServiceRoom,1..NumOfFCUsServiceRoom] of F_TRIG;  *)

  //HMIs[1..num
  HMI_Index : USINT;
  RCU_Index : USINT;
  HMI_Addresses : Array[1..NumOfHMIsServiceRoom] of USINT := [8];

  END_VAR

  if navSelect = 0 then
     lightsSelect   := 1;
     socketsSelect  := 0;

  elsif navSelect = 1 then
     lightsSelect   := 0;
     socketsSelect  := 1;
  end_if;

  HMI_Index := 7;
  RCU_Index := 5;

  if GetRemoteIPaddress(chanCode := Eth1_uni4, ethAdr := RCU_ethAdr) then
     RCUs_IPs[RCU_Index] := RCU_ethAdr.remoteIP;
  end_if;

  HMIs_Info[HMI_Index].SNo := HMI_Addresses[1];
  HMIs_Info[HMI_Index].readStAdd  := 651;
  HMIs_Info[HMI_Index].writeStAdd := 711;
  HMIs_Info[HMI_Index].readNoPoint  := SIZEOF(HMIs_DataRead[HMI_Index]) / 2;
  HMIs_Info[HMI_Index].writeNoPoint := SIZEOF(HMIs_DataWrite[HMI_Index]) / 2;

  for i := 1 to NumOfHMIsServiceRoom-1 do
    HMIs_Info[HMI_Index+i] := HMIs_Info[HMI_Index];
    HMIs_Info[HMI_Index+i].SNo := HMI_Addresses[i+1];
  end_for;

  afterRestart_TP(IN := IS_COLD_RESTART_PLC or IS_HOT_RESTART_PLC, PT := T#2s );
  afterRestart_TP_FT(CLK := afterRestart_TP.Q);

  if afterRestart_TP_FT.Q then
     SendIamServer := 1;
  end_if;

  controlRoom(RCU_ChCode := ETH1_uni4 , RCU_PingDone := RCUs_PingDone[RCU_Index],
              numOfLights := NumOfLightServiceRoom , numOfOutlets := NumOfOutletServiceRoom , numOfCurtains := 0, numOfMotionSens := NumOfMotionSensServiceRoom,
              lightsOutputDevs := lightsOutputDevs , outletOutputDevs := outletOutputDevs ,
              RCU_CH_IN := void(ETH1_uni4_IN) , LightsStatus := lightsStatusServiceRoom ,OutletsStatus := outletsStatusServiceRoom, MotionSenStatus := motionSensStatus,
              EnLights := EnLights , EnLightsAN := EnLightsAN , EnOutlets := EnOutlets ,EnOutletsAN :=EnOutletsAN ,
              SendIamServer := SendIamServer , GetAllStatus := GetAllStatus);

              //stLightsServiceRoomAN := lightsStatusServiceRoom[1];

   for i := 1 to NumOfLightServiceRoom do
       HMIs_DataWrite[HMI_Index].lightsStatus[i] := BOOL_TO_WORD(lightsStatusServiceRoom[i]);
   end_for;

   for i := 1 to NumOfOutletServiceRoom do
       HMIs_DataWrite[HMI_Index].outletsStatus[i] := BOOL_TO_WORD(outletsStatusServiceRoom[i]);
   end_for;

   for i := 1 to NumOfMotionSensServiceRoom do
       HMIs_DataWrite[HMI_Index].motionSensStatus[i] := BOOL_TO_WORD(motionSensStatus[i]);
   end_for;

   for j := 1 to NumOfHMIsServiceRoom do
     for i := 1 to NumOfLightServiceRoom do

         enLights_RT[j,i](CLK := HMIs_DataRead[HMI_Index + j - 1].enLights[i]);

         enLights_FT[j,i](CLK := HMIs_DataRead[HMI_Index + j - 1].enLights[i]);

         if enLights_RT[j,i].Q or enLights_FT[j,i].Q then
            EnLights[i] := 1;
         end_if;
     end_for;
   end_for;

   for j := 1 to NumOfHMIsServiceRoom do
     for i := 1 to NumOfOutletServiceRoom do

         enOutlets_RT[j,i](CLK := HMIs_DataRead[HMI_Index + j - 1].enOutlets[i]);

         enOutlets_FT[j,i](CLK := HMIs_DataRead[HMI_Index + j - 1].enOutlets[i]);

         if enOutlets_RT[j,i].Q or enOutlets_FT[j,i].Q then
            EnOutlets[i] := 1;
         end_if;
     end_for;
   end_for;

END_PROGRAM
